INTERFACE I_CsvRecord

METHOD PUBLIC AddBool : I_CsvRecord;
VAR_IN_OUT
	Field : BOOL;
END_VAR
END_METHOD

METHOD PUBLIC AddBoolLiteral : I_CsvRecord;
VAR_INPUT
	Field : BOOL;
END_VAR
END_METHOD

METHOD PUBLIC AddInt : I_CsvRecord;
VAR_IN_OUT
	Field : INT;
END_VAR
END_METHOD

METHOD PUBLIC AddIntLiteral : I_CsvRecord;
VAR_INPUT
	Field : INT;
END_VAR
END_METHOD

METHOD PUBLIC AddString : I_CsvRecord;
VAR_IN_OUT
	stringToWrite : STRING;
END_VAR
END_METHOD

METHOD PUBLIC AddStringLiteral : I_CsvRecord;
VAR_INPUT
	stringToWrite : STRING;
END_VAR
END_METHOD

METHOD PUBLIC EndRecord : I_CsvDocument;
END_METHOD

END_INTERFACE

(* stored: Version 1.1.0.1, ProductVersion 3.1.4024.4
   Itf I_CsvRecord: Id {1cf65c85-3558-47aa-95ce-584f0e04ec47}
   Method AddBool: Id {f0cb012e-9de8-466d-99ef-22725ead0ab5}
   Method AddBoolLiteral: Id {c7a7eeec-f740-41b7-8d23-13404ae82a63}
   Method AddInt: Id {4431b41a-890a-48fe-8dc9-dcfb2eb50447}
   Method AddIntLiteral: Id {69e63846-57ee-4558-bee9-cb0aa24ae9a9}
   Method AddString: Id {8835e7c8-d6a4-42cd-aea4-7b1de23ecf4a}
   Method AddStringLiteral: Id {7ff12bef-4cc0-46c1-8e8e-20127120ae2c}
   Method EndRecord: Id {c268a2ec-6e00-4508-83fe-0670c137b09a} *)
